TYPE "LubrMotorPump_HMI"
VERSION : 0.1
// Block: LubrMotorPump_HMI
   STRUCT
      Alarm : Bool;
      Running : Bool;
   END_STRUCT;

END_TYPE
